RoboDK station: HAMK_Robotics_station_MG400_without_tool.rdk

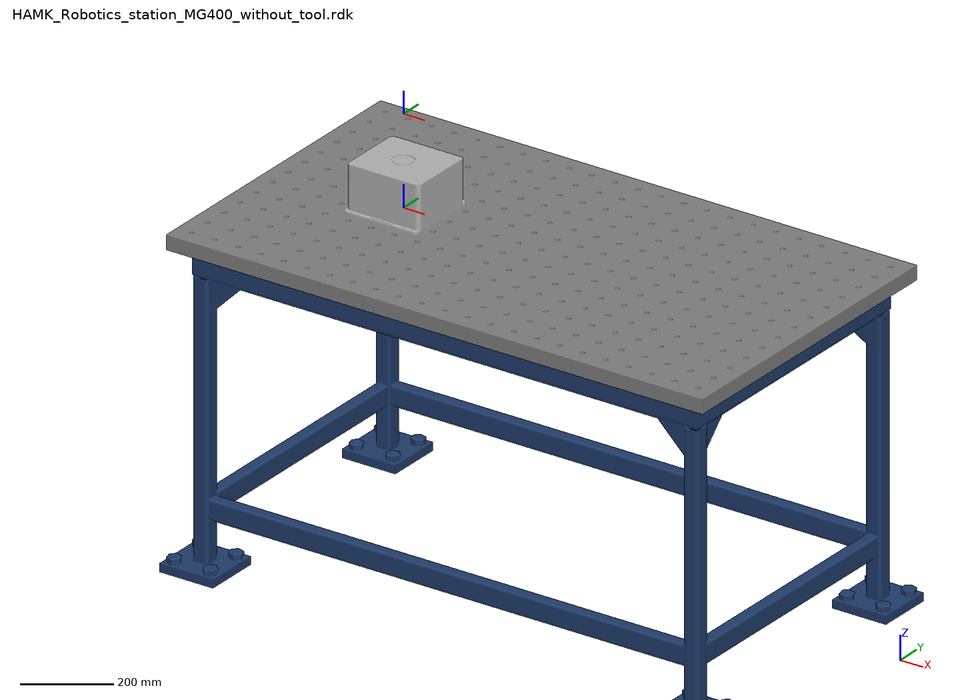
[picture v0: the station drawn from its stored meshes, robots at their saved joint values, targets as dots, program paths as lines]
Station Basic HAMK Robotics station MG400 without tool (saved by RoboDK 5.8.0). Poses are relative to the parent item; angles as X-Y-Z fixed-axis rotations.
  - frame Dobot MG400 Base at (0, 0, 0) mm
    - robot Dobot MG400: 4 axes, payload 0.5 kg, reach 393.5 mm, repeatability 0.2 mm, weight 4 kg
        joint limits [-160, -25, -25, -360] to [160, 85, 105, 360]; home [0, 0, 0, 0]; saved at [0, 0, 0, 0]
    - frame World at (0, 0, 0) mm
      - object Table 1400x800x800mm at (0, 0, 0) mm, size 1420 x 820 x 800 mm, geometry from Table-1400x800x800mm.sld
        - object HAMK logo at (360, 380, -115) mm, rotated rx 90 ry 0 rz 180 deg, size 301.4 x 100.9 x 9.4 mm, geometry from Fantastic Duup(2).stl
        - object white background at (360, 385.5, -110) mm, rotated rx 90 ry 0 rz 0 deg, size 480 x 184.8 x 2.4 mm, geometry from Fantastic Duup(3).stl
  - frame ReferenceFrameTCP at (0, 0, 223) mm
